# EPICS autosave request: gardasoftLED/PP820LED_settings.req
$(P):PERIOD
